ABB RAPID module: torques_logger.mod

MODULE torques_logger

!////////////////
!GLOBAL VARIABLES
!////////////////
!PC communication
VAR socketdev clientSocket;
VAR socketdev serverSocket;

PERS string IP;
PERS num PORT_TORQUES_LOGGER_L;
PERS tooldata currentTool;
PERS wobjdata currentWobj;
PERS num LOGGER_PERIOD;

PROC ServerCreateAndConnect(string ip, num port)
    VAR string clientIP;

    SocketCreate serverSocket;
    SocketBind serverSocket, ip, port;
    SocketListen serverSocket;
    WHILE SocketGetStatus(clientSocket) <> SOCKET_CONNECTED DO
        SocketAccept serverSocket,clientSocket \ClientAddress:=clientIP \Time:=WAIT_MAX;
        WaitTime 0.5;
    ENDWHILE
ENDPROC

PROC main()
    VAR string data;
    VAR robtarget position;
    VAR jointtarget joints;
    VAR bool connected;

    VAR string time;
    VAR clock timer;

    time:= CTime();

    connected:=FALSE;
    ServerCreateAndConnect IP, PORT_TORQUES_LOGGER_L;
    ClkStart timer;
    connected:=TRUE;

    WHILE TRUE DO

        !Cartesian Coordinates
        position := CRobT(\Tool:=currentTool \WObj:=currentWObj);
        data := "#";
        data := data + NumToStr(ClkRead(timer),2) + " ";
        data := data + NumToStr(GetMotorTorque(1),3) + " ";
        data := data + NumToStr(GetMotorTorque(2),3) + " ";
        data := data + NumToStr(GetMotorTorque(3),3) + " ";
        data := data + NumToStr(GetMotorTorque(4),3) + " ";
        data := data + NumToStr(GetMotorTorque(5),3) + " ";
        data := data + NumToStr(GetMotorTorque(6),3);
        data := data + "!";
        !End of string
        IF connected = TRUE THEN
            SocketSend clientSocket \Str:=data;
        ENDIF

        WaitTime LOGGER_PERIOD;
    ENDWHILE
    ERROR
        connected:=FALSE;
        !Closing the server
        SocketClose clientSocket;
        SocketClose serverSocket;
        !Reinitiate the server
        ServerCreateAndConnect IP, PORT_TORQUES_LOGGER_L;
        ClkReset timer;
        ClkStart timer;
        connected:= TRUE;
        RETRY;

ENDPROC

ENDMODULE
